INTERFACE IAssertionListener

METHOD OnAssertionFailed
VAR_INPUT
    AssertionMessage : T_MaxString;
    ExpectedAsString : T_MaxString;
    ActualAsString   : T_MaxString;
END_VAR
END_METHOD

PROPERTY TestName : T_MaxString
GET
END_GET
END_PROPERTY

END_INTERFACE

(* stored: Version 1.1.0.1, ProductVersion 3.1.4024.4
   Itf IAssertionListener: Id {3013ab36-1e65-0a80-2235-5faa497c56a4}
   Method OnAssertionFailed: Id {b6db4923-68d1-0c12-24c0-3d61a89106a5}
   Property TestName: Id {dc27c40f-e1a8-4651-a7e5-d85f174fe047}
   Get Get: Id {47342acb-ad81-4097-9172-3ba91aa77d32} *)
